TYPE E_DriverStatusWord :
(
	DriverStatusWord_INIT := 4641,
	DriverStatusWord_PREOP := 4659,
	DriverStatusWord_OP := 4663,
	
	MZDriverStatusWord_SwitchOnDisable := 16#40,
	MZDriverStatusWord_ReadyToSwitchOn := 16#21,
	MZDriverStatusWord_SwitchOn := 16#33,
	MZDriverStatusWord_OperationEnbale := 16#37,
	MZDriverStatusWord_Fault := 16#08
);
END_TYPE

(* stored: Version 1.1.0.1, ProductVersion 3.1.4024.12
   DUT E_DriverStatusWord: Id {13c36d80-9912-42da-8fd3-6d5f4e3aede7} *)
